FUNCTION_BLOCK "NGStatus"
VAR_INPUT
  NG_1 : Bool;
  NG_2 : Bool;
  NG_3 : Bool;
  NG_4 : Bool;
  NG_5 : Bool;
END_VAR
VAR_OUTPUT
  Status : Int;
  Ready : Bool;
END_VAR
VAR_IN_OUT
  Interlock : Array[1..10] of Bool;
END_VAR
VAR
  AlwaysOn : Bool;
  NG_Delay : Array[1..10] of TON_TIME;
  NG_DelayTime : Array[1..10] of DInt;
END_VAR
BEGIN
  // Původní jazyk: LAD
  // Zdroj XML: EXPORT/Program blocks/OP010/10_Device/29_NG/NGStatus.xml
  // --- LAD/FBD → SCL (orientační převod, jen pro revizi) ---
  // Network 1
  // --- Poznámky / omezení převodu ---
  // Síť obsahuje nepodporované prvky (ponecháno jen jako komentář): O(1)
  // SCoil UId=27: nelze určit podmínku (vstupní síť).
  // Network 2
  // --- Poznámky / omezení převodu ---
  // Síť obsahuje nepodporované prvky (ponecháno jen jako komentář): TON(5)
  // Network 3
  // --- Poznámky / omezení převodu ---
  // Síť obsahuje nepodporované prvky (ponecháno jen jako komentář): Move(1)
  // Network 4
  // --- Poznámky / omezení převodu ---
  // Síť obsahuje nepodporované prvky (ponecháno jen jako komentář): Move(1)
  // Network 5
  // --- Poznámky / omezení převodu ---
  // Síť obsahuje nepodporované prvky (ponecháno jen jako komentář): Move(1)
  // Network 6
  // --- Poznámky / omezení převodu ---
  // Síť obsahuje nepodporované prvky (ponecháno jen jako komentář): Move(1)
  // Network 7
  // --- Poznámky / omezení převodu ---
  // Síť obsahuje nepodporované prvky (ponecháno jen jako komentář): Move(1)
  // Network 8
  // --- Poznámky / omezení převodu ---
  // Síť obsahuje nepodporované prvky (ponecháno jen jako komentář): Move(1)
  // Network 9
  // --- Poznámky / omezení převodu ---
  // Síť obsahuje nepodporované prvky (ponecháno jen jako komentář): Move(1)
  // Network 10
  // --- Poznámky / omezení převodu ---
  // Síť obsahuje nepodporované prvky (ponecháno jen jako komentář): Eq(5), O(1)
  // Coil UId=42: nelze určit podmínku (vstupní síť).
END_FUNCTION_BLOCK
